Universal Robots PolyScope program: SUB_6101.urp

Program SUB_6101 (installation=GD directory=/programs/GD createdIn=5.13.0 lastSavedIn=5.13.0 robotSerialNumber=20205000017)
Calibrated DH parameters: a=[-0.000157, -0.56303, -0.236706, -0.000074, -0.000109, 0]; d=[0.181705, 47.632387, 369.599619, -417.058513, 0.119878, 0.115667]; alpha=[1.570881, -0.005074, -0.001247, 1.56886, -1.570997, 0]; deltaTheta=[0, -0.405485, 5.544791, 1.143886, -0.000009, -0.000001]
InitVariablesNode
Robot Program (runOnlyOnce=false)
  Folder ROVI_RECIPE
    If (not ROVI_RECIPE(GPII_WorkNo))
      SubPrgResult := rovi_err
      Wait Sleep waitTime=999999
  Folder ROVI_RESET
    If ( not ROVI_RESET())
      SubPrgResult := rovi_err
      Wait Sleep waitTime=999999
  Folder ROVI_CAPTURE_1
    MoveJ speed 6 deg/s, acceleration 12 deg/s^2 (useActiveTCP=false) tcp=TCP_1; feature=Base
      Switch expression=CheckMST
        Case (caseValue=0)
          Waypoint Variable (Variable): variable(featureName=Master_pos)
        Case (caseValue=1)
          Waypoint Variable (Variable): variable(featureName=Master_pos)
        Case (caseValue=2)
          Waypoint Variable (Variable): variable(featureName=Master_posL)
        Case (caseValue=3)
          Waypoint Variable (Variable): variable(featureName=Master_posR)
      SuppressedNode
        Waypoint ウェイポイント_1 (Relative): relativeFromPosition TCP in base x=-5.037 y=-329.575 z=16.043 mm, rx=-0.0235 ry=-3.1385 rz=-0.002 rad; joints [-65.945, -61.292, -135.715, -73.119, 89.887, 25.023] deg; TCP offset x=0 y=80 z=420 mm, rx=0 ry=0 rz=0 rad; TCP in base x=-3.24 y=-405.091 z=93.349 mm, rx=0.0238 ry=2.9687 rz=0.0105 rad; joints [-81.058, -70.218, -123.998, -74.522, 99.793, 10.078] deg
    Wait Sleep waitTime=3
    If ( not ROVI_CAPTURE())
      SubPrgResult := rovi_err
      Wait Sleep waitTime=999999
